// TIA Portal V20 export
DATA_BLOCK "T10 LANT I-O"   // DB1693
{ S7_Optimized_Access := 'TRUE' }
AUTHOR : SAS
// stored: AutoNumber false, IsRetainMemResEnabled true, MemoryReserve 100, RetainMemoryReserve 100
   VAR
      DI : Struct
         "E353.4" : Bool;   // (E353.4) T10-TC01: Fbk Disj Ok Ventilatoare Motoare
         "E353.5" : Bool;   // (E353.5) T10-TC01: Fbk Contactor On Ventilatoare Motoare
         "E355.6" : Bool;   // (E355.6) T10-TC01: Fbk PP1 Loading chain first pos. paralelism (1)
         "E355.7" : Bool;   // (E355.7) T10-TC01: Fbk PP2 Loading chain first pos. paralelism (2)
         "E356.2" : Bool;   // (E356.2) T10-TC01: Fbk PP1 Last position paralelism (1)
         "E356.3" : Bool;   // (E356.3) T10-TC01: Fbk PP2 Last position paralelism (2)
         "E356.4" : Bool;   // (E356.4) T10-TC01: Fbk Pos Home Step position
         "E359.3" : Bool;   // (E359.3) T10-TC:Incetinire Lant 1 Coada
         "E359.4" : Bool;   // (E359.4) T10-TC:Ultima Pozitie Lant 1 Coada
         "E359.5" : Bool;   // (E359.5) T10-TC:Incetinire Lant 2 Coada
         "E359.6" : Bool;   // (E359.6) T10-TC:Ultima Pozitie Lant 2 Coada
      END_STRUCT;
      "DO" : Struct
         "A352.2" : Bool;   // (A352.2) T10-TC01: Cmd CNT On Vent - Comanda contactor motor Vent Lant Transfer
      END_STRUCT;
      Drive : Struct
         CMD : "DRIVE_CMD_Horiz";
         STATUS { S7_SetPoint := 'True'} : "DRIVE_STATUS_Horiz";
         RD_AREA : "G120-TelegramFree8/8 READ";
         WR_AREA : "G120-TelegramFree8/8 WRITE";
      END_STRUCT;
      Encoder : Struct
         Lenght : "ENC_AUX";
         Lenght_DATA_RD { S7_SetPoint := 'True'} : "TM RD";
         Lenght_DATA_WR { S7_SetPoint := 'True'} : "TM WR";
      END_STRUCT;
   END_VAR
BEGIN
END_DATA_BLOCK
